{attribute 'call_after_init'}
FUNCTION_BLOCK FB_Sum_Test EXTENDS TcUnit.FB_TestFunctionBlock IMPLEMENTS TcUnit.I_RunnableTestFunctionBlock
VAR
	Assert : TcUnit.FB_Assert;
END_VAR

METHOD FB_init : BOOL
VAR_INPUT
	bInitRetains : BOOL; // if TRUE, the retain variables are initialized (warm start / cold start)
	bInCopyCode : BOOL;  // if TRUE, the instance afterwards gets moved into the copy code (online change)
END_VAR
SUPER^.RegisterTestFunctionBlock(THIS^);
END_METHOD

METHOD RunTests : TCUNIT.E_TestFunctionBlockRunState
TwoPlusTwoEqualsFour();
ZeroPlusZeroEqualsZero();

RunTests := TcUnit.E_TestFunctionBlockRunState.FINISHED;
END_METHOD

METHOD PRIVATE TwoPlusTwoEqualsFour
VAR
	fbSum : FB_Sum;
	nResult : UINT;
END_VAR
TEST('TwoPlusTwoEqualsFour');

fbSum(one := 2, two := 2, result => nResult);

Assert.AssertEquals_UINT(Expected := 4,
                         Actual := nResult,
                         Message := 'The calculation is not correct');
END_METHOD

METHOD PRIVATE ZeroPlusZeroEqualsZero
VAR
	fbSum : FB_Sum;
	nResult : UINT;
END_VAR
TEST('ZeroPlusZeroEqualsZero');

fbSum(one := 0, two := 0, result => nResult);

Assert.AssertEquals_UINT(Expected := 0,
                         Actual := nResult,
                         Message := 'The calculation is not correct');
END_METHOD

END_FUNCTION_BLOCK

(* stored: Version 1.1.0.1, ProductVersion 3.1.4022.12
   POU FB_Sum_Test: Id {69b661ca-5faa-43bb-8b8a-2cae13b2cfe4}, SpecialFunc None
   Method FB_init: Id {053aa1ab-2377-4f3d-852f-5268553eaca8}
   Method RunTests: Id {a311ace9-aa3c-426d-9885-bce7260e159e}
   Method TwoPlusTwoEqualsFour: Id {071ba4c3-fe0d-4b0b-be72-a320c9d403a4}
   Method ZeroPlusZeroEqualsZero: Id {ac47aa92-0e7a-4876-b0ac-7ef29219d372} *)
